TYPE ST_ItemBufferFdbk :
STRUCT
	bEmpty		: BOOL;							// Buffer is Empty
END_STRUCT
END_TYPE

(* stored: Version 1.1.0.1, ProductVersion 3.1.4024.4
   DUT ST_ItemBufferFdbk: Id {a03d18f1-8d76-4a7b-b32d-f0ec5b17012b} *)
